SYSTEM Demo
  (* Version 1.0, 2006-11-15, Goran Cengic, Chalmers *)
  DEVICE Test Device : DeviceType_not_used
    RESOURCE Test Resource : ResourceType_not_used
      FBS
        restart : E_RESTART;
        fcc : FCC;
        R3323merge : E_MERGE2;
        R3325merge : E_MERGE2;
        TT153merge : E_MERGE2;
        FIX151merge : E_MERGE2;
        rend1 : E_REND;
        rend2 : E_REND;
        rend3 : E_REND;
        coordinator : Coordinator;
        R3323coordinator : MachineCoordinator;
        R3325coordinator : MachineCoordinator;
        TT153coordinator : MachineCoordinator;
        FIX151coordinator : MachineCoordinator;
        R3323 : Machine;
        R3325 : Machine;
        TT153 : Machine;
        FIX151 : Machine;
        zone1 : Zone;
        mailbox : Mailbox;
        delay : E_DELAY;
        split1 : E_SPLIT2;
        split2 : E_SPLIT2;
        split3 : E_SPLIT2;
        split4 : E_SPLIT2;
        delay_merge : E_MERGE4;
        delay_split : E_SPLIT5;
        printd : Print;
        printr : Print;
        rend_split : E_SPLIT3;
        nomore_merge : E_MERGE2;
      END_FBS
      EVENT_CONNECTIONS
        restart.COLD TO coordinator.run;
        R3323coordinator.COPDone TO coordinator.COPDone1;
        R3325coordinator.COPDone TO coordinator.COPDone2;
        TT153coordinator.COPDone TO coordinator.COPDone3;
        FIX151coordinator.COPDone TO coordinator.COPDone4;
        coordinator.start1 TO R3323coordinator.start;
        coordinator.start2 TO R3325coordinator.start;
        coordinator.start3 TO TT153coordinator.start;
        coordinator.start4 TO FIX151coordinator.start;
        R3323coordinator.send TO mailbox.sendMC1;
        R3325coordinator.send TO mailbox.sendMC2;
        TT153coordinator.send TO mailbox.sendMC3;
        FIX151coordinator.send TO mailbox.sendMC4;
        R3323.send TO mailbox.sendM1;
        R3325.send TO mailbox.sendM2;
        TT153.send TO mailbox.sendM3;
        FIX151.send TO mailbox.sendM4;
        zone1.send TO mailbox.sendZ1;
        mailbox.toMC1 TO R3323coordinator.receive;
        mailbox.toMC2 TO R3325coordinator.receive;
        mailbox.toMC3 TO TT153coordinator.receive;
        mailbox.toMC4 TO FIX151coordinator.receive;
        mailbox.toM1 TO R3323.receive;
        mailbox.toM2 TO R3325.receive;
        mailbox.toM3 TO TT153.receive;
        mailbox.toM4 TO FIX151.receive;
        mailbox.toZ1 TO zone1.receive;
        R3323.startOperation TO fcc.startOperationM1;
        R3325.startOperation TO fcc.startOperationM2;
        TT153.startOperation TO fcc.startOperationM3;
        FIX151.startOperation TO fcc.startOperationM4;
        fcc.finishedOperationM1 TO R3323.finishedOperation;
        fcc.finishedOperationM2 TO R3325.finishedOperation;
        fcc.finishedOperationM3 TO TT153.finishedOperation;
        fcc.finishedOperationM4 TO FIX151.finishedOperation;
        R3323coordinator.noMoreEvents TO R3323merge.EI1;
        R3325coordinator.noMoreEvents TO R3325merge.EI1;
        TT153coordinator.noMoreEvents TO TT153merge.EI1;
        FIX151coordinator.noMoreEvents TO FIX151merge.EI1;
        R3323.noMoreEvents TO R3323merge.EI2;
        R3325.noMoreEvents TO R3325merge.EI2;
        TT153.noMoreEvents TO TT153merge.EI2;
        FIX151.noMoreEvents TO FIX151merge.EI2;
        R3323merge.EO TO split1.EI;
        R3325merge.EO TO split2.EI;
        TT153merge.EO TO split3.EI;
        FIX151merge.EO TO split4.EI;
        split1.EO1 TO rend1.EI1;
        split2.EO1 TO rend1.EI2;
        split3.EO1 TO rend2.EI1;
        split4.EO1 TO rend2.EI2;
        rend1.EO TO rend3.EI1;
        rend2.EO TO rend3.EI2;
        rend3.EO TO rend_split.EI;
        split1.EO2 TO delay_merge.EI1;
        split2.EO2 TO delay_merge.EI2;
        split3.EO2 TO delay_merge.EI3;
        split4.EO2 TO delay_merge.EI4;
        delay_merge.EO TO delay.START;
        rend_split.EO1 TO delay.STOP;
        rend_split.EO2 TO nomore_merge.EI1;
        rend_split.EO3 TO printr.PRINT;
        delay.EO TO delay_split.EI;
        delay_split.EO1 TO nomore_merge.EI2;
        delay_split.EO2 TO rend1.R;
        delay_split.EO3 TO rend2.R;
        delay_split.EO4 TO rend3.R;
        delay_split.EO5 TO printd.PRINT;
        nomore_merge.EO TO fcc.noMoreEvents;
      END_CONNECTIONS
      DATA_CONNECTIONS
        App Delay triggered TO printd.TEXT;
        App Rendesvouz triggered TO printr.TEXT;
        1000 TO delay.DT;
        R3323coordinator.machineName TO coordinator.machineName1;
        R3323coordinator.performed TO coordinator.performed1;
        R3325coordinator.machineName TO coordinator.machineName2;
        R3325coordinator.performed TO coordinator.performed2;
        TT153coordinator.machineName TO coordinator.machineName3;
        TT153coordinator.performed TO coordinator.performed3;
        FIX151coordinator.machineName TO coordinator.machineName4;
        FIX151coordinator.performed TO coordinator.performed4;
        R3323coordinator.outMessage TO mailbox.inMessageMC1;
        mailbox.outMessageMC1 TO R3323coordinator.inMessage;
        R3325coordinator.outMessage TO mailbox.inMessageMC2;
        mailbox.outMessageMC2 TO R3325coordinator.inMessage;
        TT153coordinator.outMessage TO mailbox.inMessageMC3;
        mailbox.outMessageMC3 TO TT153coordinator.inMessage;
        FIX151coordinator.outMessage TO mailbox.inMessageMC4;
        mailbox.outMessageMC4 TO FIX151coordinator.inMessage;
        R3323.outMessage TO mailbox.inMessageM1;
        mailbox.outMessageM1 TO R3323.inMessage;
        R3325.outMessage TO mailbox.inMessageM2;
        mailbox.outMessageM2 TO R3325.inMessage;
        TT153.outMessage TO mailbox.inMessageM3;
        mailbox.outMessageM3 TO TT153.inMessage;
        FIX151.outMessage TO mailbox.inMessageM4;
        mailbox.outMessageM4 TO FIX151.inMessage;
        zone1.outMessage TO mailbox.inMessageZ1;
        mailbox.outMessageZ1 TO zone1.inMessage;
        R3323.outOperation TO fcc.inOperationM1;
        R3325.outOperation TO fcc.inOperationM2;
        TT153.outOperation TO fcc.inOperationM3;
        FIX151.outOperation TO fcc.inOperationM4;
        fcc.outOperationM1 TO R3323.inOperation;
        fcc.outOperationM2 TO R3325.inOperation;
        fcc.outOperationM3 TO TT153.inOperation;
        fcc.outOperationM4 TO FIX151.inOperation;
      END_CONNECTIONS
    END_RESOURCE
  END_DEVICE
END_SYSTEM
